TYPE stTarget3D EXTENDS stTarget :
STRUCT
	pose : stPose3D;
END_STRUCT
END_TYPE

(* stored: Version 1.1.0.1, ProductVersion 3.1.4026.18
   DUT stTarget3D: Id {c1b2c3d4-4444-4444-4444-444444444444} *)
